TYPE TempSensor_SelectStruct :
STRUCT
	SensorValue: STRING(255);
	SampleNr: DINT;
	Time_: DT;
	SensorID: DINT;
END_STRUCT
END_TYPE

(* stored: Version 1.1.0.1
   DUT TempSensor_SelectStruct: Id {f86cf38e-752e-4498-893f-2e6b28d104c2} *)
